// Block: PPrgArchive5

DATA_BLOCK PPrgArchive5
VERSION : 0.1
   NON_RETAIN
   VAR
      PRG : Array[401..500] of PPrg_Data;
   END_VAR

BEGIN
   // No initialization required
END_DATA_BLOCK
